FUNCTION_BLOCK EL1814
VAR
	_io : EL1xx4_Data;
	{attribute addProperty Name "WcState"}
	_wcState : WcStateInputToggle;
	{attribute addProperty Name "Info data"}
	_infoData : InfoDataBase;
END_VAR

PROPERTY IO : REFERENCE TO EL1xx4_Data
GET
IO REF= _io;
END_GET
END_PROPERTY

PROPERTY WcState : REFERENCE TO WcStateInputToggle
GET
WcState REF= _wcState;
END_GET
END_PROPERTY

END_FUNCTION_BLOCK

(* stored: Version 1.1.0.1, ProductVersion 3.1.4024.9
   POU EL1814: Id {c51c1c69-d00f-0989-0641-60dfc5ea555a}, SpecialFunc None
   Property IO: Id {52cdbffb-5a44-09aa-1b4a-74f4a644f28e}
   Get Get: Id {75fb9826-0414-0c98-0ff0-d4e604aab583}
   Property WcState: Id {6606b916-6571-0f2d-215e-565ed7eaa69e}
   Get Get: Id {48cb6512-486d-024a-1f56-819489c177c8} *)
